// TwinCAT 3 PLC project MotionRail
// ProgramVersion: 3.1.4022.3
// libraries:
//   Tc2_MC2, * (Beckhoff Automation GmbH)
//   Tc2_Standard, * (Beckhoff Automation GmbH)
//   Tc2_System, * (Beckhoff Automation GmbH)
//   Tc3_Module, * (Beckhoff Automation GmbH)
// project tree:
//   / PlcTask.TcTTO
//   POUs/ FB_MicroStepCountTest.TcPOU, FB_MicroStepWalkTest.TcPOU, MAIN.TcPOU, FB_Tuning.TcPOU
// real-time tasks:
//   TASK PlcTask: cycle T#10ms, priority 20, ADS port 350
// motion (NC):
//   TASK NC-Task 1 SAF: cycle T#2ms, priority 4, ADS port 501
//   TASK NC-Task 1 SVB: cycle T#10ms, priority 8, ADS port 511
//   AXIS Axis 1 (id 1)
//     Dynamic: AccelerationMaximum=5, DecelerationMaximum=5, Acceleration=5, Deceleration=5, Jerk=5, DelayTime=0.008
//     Velo: Maximum=20
//     OtherSettings: AllowMotionCmdToSlave=true
//     encoder EncType=29
//       EncPara: ScaleFactorNumerator=5e-005, MaxCount=#xffffffff
//         SoftEndMinControl: Enable=true, Range=25
//         SoftEndMaxControl: Enable=true, Range=110
//         Inc: RefSoftSyncMask=#x0000ffff
//     drive DrvType=24
//       Analog: VeloReferenz=50, ScaleFactorActTorque=0.1
//       TimeComp: TaskDelayCycles=1
//     controller CtrType=2
//       CtrPara: PriorControlFactor=1
//         PosDiffControl: Range=0.1
//         PID: PosKp=20, PosExtKp=20, DeadBandPosition=0.000195
//         Observer: BandWidth=20
//   AXIS Axis 2 (id 2)
//     Dynamic: DelayTime=0.008
//     Velo: Maximum=5
//     OtherSettings: AllowMotionCmdToSlave=true
//     encoder EncType=4
//       EncPara: ScaleFactorNumerator=0.0001984375, MaxCount=#x0000ffff
//         Inc: RefMode=2, RefSoftSyncMask=#x0000ffff
//     drive DrvType=24
//       Analog: VeloReferenz=25.4, ScaleFactorActTorque=0.1
//       TimeComp: TaskDelayCycles=1
//     controller CtrType=1
//       CtrPara: PriorControlFactor=1
//         PosDiffControl: Range=0.635
//         Observer: BandWidth=20
//   AXIS Axis 3 (id 3)
//     Dynamic: DelayTime=0.008
//     Velo: Maximum=5
//     OtherSettings: AllowMotionCmdToSlave=true
//     encoder EncType=4
//       EncPara: ScaleFactorNumerator=0.0001984375, MaxCount=#x0000ffff
//         Inc: RefSoftSyncMask=#x0000ffff
//     drive DrvType=24
//       Analog: VeloReferenz=24.80437, ScaleFactorActTorque=0.1
//       TimeComp: TaskDelayCycles=1
//     controller CtrType=1
//       CtrPara: PriorControlFactor=1
//         PosDiffControl: Range=0.635
//         Observer: BandWidth=20
//   AXIS Axis 4 (id 4)
//     Dynamic: AccelerationMaximum=1000, DecelerationMaximum=1000, Acceleration=10, Deceleration=10, Jerk=100, DelayTime=0.008
//     Velo: RefSearch=1, RefSync=1, SlowManual=5, FastManual=5, Maximum=9
//     TargetPosControl: Range=0.001, Time=0.2
//     OtherSettings: AllowMotionCmdToSlave=true, PulseDistancePos=2, PulseDistanceNeg=2
//     encoder EncType=29
//       EncPara: ScaleFactorNumerator=5e-005, MaxCount=#xffffffff, ReferenceSystem=1
//         SoftEndMinControl: Enable=true, Range=5
//         SoftEndMaxControl: Enable=true, Range=60
//         Inc: RefSoftSyncMask=#x0000ffff
//     drive DrvType=24
//       Analog: VeloReferenz=25.4, ScaleFactorActTorque=0.1
//       TimeComp: TaskDelayCycles=1
//     controller CtrType=2
//       CtrPara: PriorControlFactor=1
//         PosDiffControl: Range=0.1
//         PID: PosKp=20, PosExtKp=5, DeadBandPosition=0.0001
//         Observer: BandWidth=20
// I/O:
//   DEVICE Device 1 (EtherCAT), AmsNetId 5.54.18.124.2.1
//     Term 1 (EK1200) [EK1200-5000 EtherCAT Power supply (2A E-Bus)]
//       Term 2 (EL7041) [EL7041 1Ch. Stepper motor output stage (50V, 5A)]
//       Term 3 (EL1004) [EL1004 4Ch. Dig. Input 24V, 3ms]
//       Term 4 (EL2008) [EL2008 8Ch. Dig. Output 24V, 0.5A]
//       Term 5 (EL5042) [EL5042 2Ch. BiSS-C Encoder]
//       Term 6 (EL7031) [EL7031 1Ch. Stepper motor output stage (24V, 1.5A)]
//       Term 7 (EL6001) [EL6001 Interface (RS232)]
//       Term 8 (EL7041-1000) [EL7041-1000 1Ch. Stepper motor output stage (50V, 5A, standard)]
//       Term 9 (EL5042) [EL5042 2Ch. BiSS-C Encoder]
//       Term 10 (EL7041) [EL7041 1Ch. Stepper motor output stage (50V, 5A)]
//       Term 11 (EL5042) [EL5042 2Ch. BiSS-C Encoder]
//       Term 12 (EL9011)
// variable links:
//   (this object) <-> Device 1 (EtherCAT)/Term 1 (EK1200)/Term 2 (EL7041)
//     Drive/Inputs/In/nState1 @bit 3 <-> STM Status/Status/Error
//     Drive/Inputs/In/nState1 @bit 5 <-> STM Status/Status/Moving negative
//     Drive/Inputs/In/nState1 @bit 4 <-> STM Status/Status/Moving positive
//     Drive/Inputs/In/nState1 @bit 1 <-> STM Status/Status/Ready
//     Drive/Inputs/In/nState1 <-> STM Status/Status/Ready to enable
//     Drive/Inputs/In/nState1 @bit 6 <-> STM Status/Status/Torque reduced
//     Drive/Inputs/In/nState1 @bit 2 <-> STM Status/Status/Warning
//     Drive/Inputs/In/nState2 @bit 3 <-> STM Status/Status/Digital input 1
//     Drive/Inputs/In/nState2 @bit 4 <-> STM Status/Status/Digital input 2
//     Drive/Inputs/In/nState4 @bit 1 <-> WcState/InputToggle
//     Drive/Inputs/In/nState4 <-> WcState/WcState
//     Drive/Outputs/Out/nCtrl1 <-> STM Control/Control/Enable
//     Drive/Outputs/Out/nCtrl1 @bit 2 <-> STM Control/Control/Reduce torque
//     Drive/Outputs/Out/nCtrl1 @bit 1 <-> STM Control/Control/Reset
//     Drive/Outputs/Out/nDataOut2[0] <-> STM Velocity/Velocity
//   (this object) <-> Device 1 (EtherCAT)/Term 1 (EK1200)/Term 5 (EL5042)
//     Enc/Inputs/In/nComState @bit 1 <-> WcState/InputToggle
//     Enc/Inputs/In/nComState <-> WcState/WcState
//     Enc/Inputs/In/nDataIn1 <-> FB Inputs Channel 1/Position
//     Enc/Inputs/In/nState1 @bit 12 <-> FB Inputs Channel 1/Status/Diag
//     Enc/Inputs/In/nState1 @bit 1 <-> FB Inputs Channel 1/Status/Error
//     Enc/Inputs/In/nState1 @bit 14 <-> FB Inputs Channel 1/Status/Input cycle counter
//     Enc/Inputs/In/nState1 @bit 2 <-> FB Inputs Channel 1/Status/Ready
//     Enc/Inputs/In/nState1 @bit 13 <-> FB Inputs Channel 1/Status/TxPDO State
//     Enc/Inputs/In/nState1 <-> FB Inputs Channel 1/Status/Warning
//   (this object) <-> Device 1 (EtherCAT)/Term 1 (EK1200)/Term 6 (EL7031)
//     Drive/Inputs/In/nState1 @bit 3 <-> STM Status/Status/Error
//     Drive/Inputs/In/nState1 @bit 5 <-> STM Status/Status/Moving negative
//     Drive/Inputs/In/nState1 @bit 4 <-> STM Status/Status/Moving positive
//     Drive/Inputs/In/nState1 @bit 1 <-> STM Status/Status/Ready
//     Drive/Inputs/In/nState1 <-> STM Status/Status/Ready to enable
//     Drive/Inputs/In/nState1 @bit 6 <-> STM Status/Status/Torque reduced
//     Drive/Inputs/In/nState1 @bit 2 <-> STM Status/Status/Warning
//     Drive/Inputs/In/nState2 @bit 3 <-> STM Status/Status/Digital input 1
//     Drive/Inputs/In/nState2 @bit 4 <-> STM Status/Status/Digital input 2
//     Drive/Inputs/In/nState2 @bit 5 <-> STM Status/Status/Sync error
//     Drive/Inputs/In/nState2 @bit 7 <-> STM Status/Status/TxPDO Toggle
//     Drive/Inputs/In/nState4 @bit 1 <-> WcState/InputToggle
//     Drive/Inputs/In/nState4 <-> WcState/WcState
//     Drive/Outputs/Out/nCtrl1 <-> STM Control/Control/Enable
//     Drive/Outputs/Out/nCtrl1 @bit 2 <-> STM Control/Control/Reduce torque
//     Drive/Outputs/Out/nCtrl1 @bit 1 <-> STM Control/Control/Reset
//     Drive/Outputs/Out/nDataOut2[0] <-> STM Velocity/Velocity
//     Enc/Inputs/In/nDataIn1[0] <-> ENC Status compact/Counter value
//     Enc/Inputs/In/nDataIn2[0] <-> ENC Status compact/Latch value
//     Enc/Inputs/In/nState1 @bit 4 <-> ENC Status compact/Status/Counter overflow
//     Enc/Inputs/In/nState1 @bit 3 <-> ENC Status compact/Status/Counter underflow
//     Enc/Inputs/In/nState1 @bit 1 <-> ENC Status compact/Status/Latch extern valid
//     Enc/Inputs/In/nState1 @bit 2 <-> ENC Status compact/Status/Set counter done
//     Enc/Inputs/In/nState2 @bit 4 <-> ENC Status compact/Status/Status of extern latch
//     Enc/Inputs/In/nState2 @bit 5 <-> ENC Status compact/Status/Sync error
//     Enc/Inputs/In/nState2 @bit 7 <-> ENC Status compact/Status/TxPDO Toggle
//     Enc/Inputs/In/nState4 @bit 1 <-> WcState/InputToggle
//     Enc/Inputs/In/nState4 <-> WcState/WcState
//     Enc/Outputs/Out/nCtrl1 @bit 3 <-> ENC Control compact/Control/Enable latch extern on negative edge
//     Enc/Outputs/Out/nCtrl1 @bit 1 <-> ENC Control compact/Control/Enable latch extern on positive edge
//     Enc/Outputs/Out/nCtrl1 @bit 2 <-> ENC Control compact/Control/Set counter
//     Enc/Outputs/Out/nDataOut1[0] <-> ENC Control compact/Set counter value
//   (this object) <-> Device 1 (EtherCAT)/Term 1 (EK1200)/Term 8 (EL7041-1000)
//     Drive/Inputs/In/nState1 @bit 3 <-> STM Status/Status/Error
//     Drive/Inputs/In/nState1 @bit 5 <-> STM Status/Status/Moving negative
//     Drive/Inputs/In/nState1 @bit 4 <-> STM Status/Status/Moving positive
//     Drive/Inputs/In/nState1 @bit 1 <-> STM Status/Status/Ready
//     Drive/Inputs/In/nState1 <-> STM Status/Status/Ready to enable
//     Drive/Inputs/In/nState1 @bit 6 <-> STM Status/Status/Torque reduced
//     Drive/Inputs/In/nState1 @bit 2 <-> STM Status/Status/Warning
//     Drive/Inputs/In/nState2 @bit 3 <-> STM Status/Status/Digital input 1
//     Drive/Inputs/In/nState2 @bit 4 <-> STM Status/Status/Digital input 2
//     Drive/Inputs/In/nState2 @bit 5 <-> STM Status/Status/Sync error
//     Drive/Inputs/In/nState2 @bit 7 <-> STM Status/Status/TxPDO Toggle
//     Drive/Inputs/In/nState4 @bit 1 <-> WcState/InputToggle
//     Drive/Inputs/In/nState4 <-> WcState/WcState
//     Drive/Outputs/Out/nCtrl1 <-> STM Control/Control/Enable
//     Drive/Outputs/Out/nCtrl1 @bit 2 <-> STM Control/Control/Reduce torque
//     Drive/Outputs/Out/nCtrl1 @bit 1 <-> STM Control/Control/Reset
//     Drive/Outputs/Out/nDataOut2[0] <-> STM Velocity/Velocity
//     Enc/Inputs/In/nDataIn1[0] <-> ENC Status compact/Counter value
//     Enc/Inputs/In/nDataIn2[0] <-> ENC Status compact/Latch value
//     Enc/Inputs/In/nState1 @bit 4 <-> ENC Status compact/Status/Counter overflow
//     Enc/Inputs/In/nState1 @bit 3 <-> ENC Status compact/Status/Counter underflow
//     Enc/Inputs/In/nState1 @bit 7 <-> ENC Status compact/Status/Extrapolation stall
//     Enc/Inputs/In/nState1 <-> ENC Status compact/Status/Latch C valid
//     Enc/Inputs/In/nState1 @bit 1 <-> ENC Status compact/Status/Latch extern valid
//     Enc/Inputs/In/nState1 @bit 2 <-> ENC Status compact/Status/Set counter done
//     Enc/Inputs/In/nState2 @bit 4 <-> ENC Status compact/Status/Status of extern latch
//     Enc/Inputs/In/nState2 <-> ENC Status compact/Status/Status of input A
//     Enc/Inputs/In/nState2 @bit 1 <-> ENC Status compact/Status/Status of input B
//     Enc/Inputs/In/nState2 @bit 2 <-> ENC Status compact/Status/Status of input C
//     Enc/Inputs/In/nState2 @bit 5 <-> ENC Status compact/Status/Sync error
//     Enc/Inputs/In/nState2 @bit 7 <-> ENC Status compact/Status/TxPDO Toggle
//     Enc/Inputs/In/nState4 @bit 1 <-> WcState/InputToggle
//     Enc/Inputs/In/nState4 <-> WcState/WcState
//     Enc/Outputs/Out/nCtrl1 <-> ENC Control compact/Control/Enable latch C
//     Enc/Outputs/Out/nCtrl1 @bit 3 <-> ENC Control compact/Control/Enable latch extern on negative edge
//     Enc/Outputs/Out/nCtrl1 @bit 1 <-> ENC Control compact/Control/Enable latch extern on positive edge
//     Enc/Outputs/Out/nCtrl1 @bit 2 <-> ENC Control compact/Control/Set counter
//     Enc/Outputs/Out/nDataOut1[0] <-> ENC Control compact/Set counter value
//   (this object) <-> Device 1 (EtherCAT)/Term 1 (EK1200)/Term 10 (EL7041)
//     Drive/Inputs/In/nState1 @bit 3 <-> STM Status/Status/Error
//     Drive/Inputs/In/nState1 @bit 5 <-> STM Status/Status/Moving negative
//     Drive/Inputs/In/nState1 @bit 4 <-> STM Status/Status/Moving positive
//     Drive/Inputs/In/nState1 @bit 1 <-> STM Status/Status/Ready
//     Drive/Inputs/In/nState1 <-> STM Status/Status/Ready to enable
//     Drive/Inputs/In/nState1 @bit 6 <-> STM Status/Status/Torque reduced
//     Drive/Inputs/In/nState1 @bit 2 <-> STM Status/Status/Warning
//     Drive/Inputs/In/nState2 @bit 3 <-> STM Status/Status/Digital input 1
//     Drive/Inputs/In/nState2 @bit 4 <-> STM Status/Status/Digital input 2
//     Drive/Inputs/In/nState2 @bit 5 <-> STM Status/Status/Sync error
//     Drive/Inputs/In/nState2 @bit 7 <-> STM Status/Status/TxPDO Toggle
//     Drive/Inputs/In/nState4 @bit 1 <-> WcState/InputToggle
//     Drive/Inputs/In/nState4 <-> WcState/WcState
//     Drive/Outputs/Out/nCtrl1 <-> STM Control/Control/Enable
//     Drive/Outputs/Out/nCtrl1 @bit 2 <-> STM Control/Control/Reduce torque
//     Drive/Outputs/Out/nCtrl1 @bit 1 <-> STM Control/Control/Reset
//     Drive/Outputs/Out/nDataOut2[0] <-> STM Velocity/Velocity
//   (this object) <-> Device 1 (EtherCAT)/Term 1 (EK1200)/Term 11 (EL5042)
//     Enc/Inputs/In/nComState @bit 1 <-> WcState/InputToggle
//     Enc/Inputs/In/nComState <-> WcState/WcState
//     Enc/Inputs/In/nDataIn1 <-> FB Inputs Channel 1/Position
//     Enc/Inputs/In/nState1 @bit 12 <-> FB Inputs Channel 1/Status/Diag
//     Enc/Inputs/In/nState1 @bit 1 <-> FB Inputs Channel 1/Status/Error
//     Enc/Inputs/In/nState1 @bit 14 <-> FB Inputs Channel 1/Status/Input cycle counter
//     Enc/Inputs/In/nState1 @bit 2 <-> FB Inputs Channel 1/Status/Ready
//     Enc/Inputs/In/nState1 @bit 13 <-> FB Inputs Channel 1/Status/TxPDO State
//     Enc/Inputs/In/nState1 <-> FB Inputs Channel 1/Status/Warning
//   MotionRail Instance <-> Device 1 (EtherCAT)/Term 1 (EK1200)/Term 10 (EL7041)
//     PlcTask Inputs/MAIN.bLimBwd4 <-> STM Status/Status/Digital input 2
//     PlcTask Inputs/MAIN.bLimFwd4 <-> STM Status/Status/Digital input 1
//   MotionRail Instance <-> Device 1 (EtherCAT)/Term 1 (EK1200)/Term 11 (EL5042)
//     PlcTask Inputs/MAIN.nRawCount4 <-> FB Inputs Channel 1/Position
//   MotionRail Instance <-> Device 1 (EtherCAT)/Term 1 (EK1200)/Term 2 (EL7041)
//     PlcTask Inputs/MAIN.bLimBwd1 <-> STM Status/Status/Digital input 2
//     PlcTask Inputs/MAIN.bLimFwd1 <-> STM Status/Status/Digital input 1
//   MotionRail Instance <-> Device 1 (EtherCAT)/Term 1 (EK1200)/Term 3 (EL1004)
//     PlcTask Inputs/MAIN.bHome1 <-> Channel 1/Input
//   MotionRail Instance <-> Device 1 (EtherCAT)/Term 1 (EK1200)/Term 4 (EL2008)
//     PlcTask Outputs/MAIN.bBrake1 <-> Channel 1/Output
//   MotionRail Instance <-> Device 1 (EtherCAT)/Term 1 (EK1200)/Term 5 (EL5042)
//     PlcTask Inputs/MAIN.fEnc2Raw <-> FB Inputs Channel 2/Position
//     PlcTask Inputs/MAIN.nRawCount1 <-> FB Inputs Channel 1/Position
//     PlcTask Inputs/MAIN.nRawCount2 <-> FB Inputs Channel 2/Position
//   MotionRail Instance <-> Device 1 (EtherCAT)/Term 1 (EK1200)/Term 6 (EL7031)
//     PlcTask Inputs/MAIN.bLimBwd2 <-> STM Status/Status/Digital input 2
//     PlcTask Inputs/MAIN.bLimFwd2 <-> STM Status/Status/Digital input 1
//   MotionRail Instance <-> Device 1 (EtherCAT)/Term 1 (EK1200)/Term 8 (EL7041-1000)
//     PlcTask Inputs/MAIN.bLimBwd3 <-> STM Status/Status/Digital input 2
//     PlcTask Inputs/MAIN.bLimFwd3 <-> STM Status/Status/Digital input 1
//   MotionRail Instance <-> Device 1 (EtherCAT)/Term 1 (EK1200)/Term 9 (EL5042)
//     PlcTask Inputs/MAIN.nRawCount3 <-> FB Inputs Channel 1/Position
//   MotionRail Instance <-> NC-Task 1 SAF/Axes/Axis 1
//     PlcTask Inputs/MAIN.Axis1.NcToPlc <-> Outputs/ToPlc
//     PlcTask Outputs/MAIN.Axis1.PlcToNc <-> Inputs/FromPlc
//   MotionRail Instance <-> NC-Task 1 SAF/Axes/Axis 2
//     PlcTask Inputs/MAIN.Axis2.NcToPlc <-> Outputs/ToPlc
//     PlcTask Outputs/MAIN.Axis2.PlcToNc <-> Inputs/FromPlc
//   MotionRail Instance <-> NC-Task 1 SAF/Axes/Axis 3
//     PlcTask Inputs/MAIN.Axis3.NcToPlc <-> Outputs/ToPlc
//     PlcTask Outputs/MAIN.Axis3.PlcToNc <-> Inputs/FromPlc
//   MotionRail Instance <-> NC-Task 1 SAF/Axes/Axis 4
//     PlcTask Inputs/MAIN.Axis4.NcToPlc <-> Outputs/ToPlc
//     PlcTask Outputs/MAIN.Axis4.PlcToNc <-> Inputs/FromPlc

CONFIGURATION MotionRail
    RESOURCE PLC ON TwinCAT3
        TASK PlcTask(INTERVAL := T#10ms, PRIORITY := 20);
        PROGRAM MAIN WITH PlcTask : MAIN;
    END_RESOURCE
END_CONFIGURATION

// ---- POUs/MAIN.TcPOU
PROGRAM MAIN
VAR
	Axis1: AXIS_REF;
	fbPower1: MC_POWER;
	bEnable1: BOOL := FALSE;
	bLimFwd1 AT %I*: BOOL;
	bLimBwd1 AT %I*: BOOL;
	bHome1 AT %I*: BOOL;
	bBrake1 AT %Q*: BOOL;
	fDeadband1: LREAL;
	fInvDeadband1: LREAL;
	nRawCount1 AT %I*: ULINT;
	
	Axis2: AXIS_REF;
	fbPower2: MC_POWER;
	bEnable2: BOOL := FALSE;
	bLimFwd2 AT %I*: BOOL;
	bLimBwd2 AT %I*: BOOL;
	bBrake2 AT %Q*: BOOL;
	fEnc2Raw AT %I*: LREAL;
	fDeadband2: LREAL;
	fInvDeadband2: LREAL;	
	nRawCount2 AT %I*: ULINT;
	
	Axis3: AXIS_REF;
	fbPower3: MC_POWER;
	bEnable3: BOOL := FALSE;
	bLimFwd3 AT %I*: BOOL;
	bLimBwd3 AT %I*: BOOL;
	bBrake3 AT %Q*: BOOL;
	fDeadband3: LREAL;
	fInvDeadband3: LREAL;
	nRawCount3 AT %I*: ULINT;
	
	Axis4: AXIS_REF;
	fbPower4: MC_POWER;
	bEnable4: BOOL := FALSE;
	bLimFwd4 AT %I*: BOOL;
	bLimBwd4 AT %I*: BOOL;
	bBrake4 AT %Q*: BOOL;
	fDeadband4: LREAL;
	fInvDeadband4: LREAL;
	nRawCount4 AT %I*: ULINT;
	
	bRefZero: BOOL;

	bDoTest: BOOL := FALSE;
	fbMicroWalkTest: FB_MicroStepWalkTest;
END_VAR

// Axis 1 is the standard circular motor connector + renishaw default pinout on the first channel of the first 5042
Axis1.ReadStatus();
fbPower1(Axis:=Axis1,
	Enable:=bEnable1,
	Enable_Positive:=bLimFwd1 OR TRUE,
	Enable_Negative:=bLimBwd1);
bBrake1 := Axis1.Status.ControlLoopClosed;
fDeadband1 := 0.000390625 / 2;
fInvDeadband1 := -fDeadband1;

// Axis 2 is the all-in-one motor/encoder connector on the second channel of the first 5042
Axis2.ReadStatus();
fbPower2(Axis:=Axis2,
	Enable:=bEnable2,
	Enable_Positive:=NOT bLimFwd2 OR TRUE,
	Enable_Negative:=NOT bLimBwd2 OR TRUE);
bBrake2 := Axis2.Status.ControlLoopClosed;

// Axis 3 is the stage with the magnetic encoder going to the first channel of the second 5042
Axis3.ReadStatus();
fbPower3(Axis:=Axis3,
	Enable:=bEnable3,
	Enable_Positive:=NOT bLimFwd3 OR TRUE,
	Enable_Negative:=NOT bLimBwd3 OR TRUE);
bBrake3 := Axis3.Status.ControlLoopClosed;

// Axis 4 is Alex's stage, going to the 4th drive and into the first channel of the third 5042
Axis4.ReadStatus();
fbPower4(Axis:=Axis4,
	Enable:=bEnable4,
	Enable_Positive:=NOT bLimFwd4 OR TRUE,
	Enable_Negative:=NOT bLimBwd4 OR TRUE);
bBrake4 := Axis4.Status.ControlLoopClosed;
fDeadband4 := 0.0001984375 / 2;
fInvDeadband4 := -1 * fDeadband4;

fbMicroWalkTest(bExecute:=bDoTest,
	nSteps:=1000,
	fDeadband:=fDeadband4 + 0.000025,
	fLowerBound:=10,
	fUpperBound:=55,
	fVelocity:=1,
	tSettleTime:=T#5S,
	Axis:=Axis4);

END_PROGRAM

// ---- POUs/FB_MicroStepWalkTest.TcPOU
FUNCTION_BLOCK FB_MicroStepWalkTest
VAR_INPUT
	bExecute: BOOL;
	nSteps: UINT;
	fDeadband: LREAL;
	fLowerBound: LREAL;
	fUpperBound: LREAL;
	fVelocity: LREAL;
	tSettleTime: TIME;
END_VAR
VAR_OUTPUT
	nGood: UINT;
	nBad: UINT;
	fPercent: LREAL;
	fAvgErr: LREAL;
	fMaxErr: LREAL;
	fMinErr: LREAL := 9001;
END_VAR
VAR_IN_OUT
	Axis: AXIS_REF;
END_VAR
VAR
	fbRand: DRAND;
	fbMove: MC_MoveAbsolute;
	fbSettleTimer: TON;
	bDoMove: BOOL;
	fGoal: LREAL;
	fStepErr: LREAL;
	fTotalErr: LREAL;
	nStepCounter: UINT;
END_VAR

// Moves to random positions and see how close we get to each one
// Pick random numbers from 0 to 1
fbRand(Seed:=UINT_TO_INT(nSteps));
// Latch a new random goal if we aren't moving
IF NOT bDoMove THEN
	fGoal := fbRand.Num * (fUpperBound - fLowerBound) + fLowerBound;
END_IF
// Motion FB
fbMove(Axis:=Axis,
	Execute:=bDoMove,
	Position:=fGoal,
	Velocity:=fVelocity);
// Settle time
fbSettleTimer(IN:=fbMove.Done,
	PT:=tSettleTime);
// Re-enable the move for next cycle
bDoMove := bExecute AND nStepCounter < nSteps;
// Check results
IF fbSettleTimer.Q THEN
	fStepErr := ABS(Axis.NcToPlc.PosDiff);
	IF fStepErr <= fDeadband THEN
		nGood := nGood + 1;
	ELSE
		nBad := nBad + 1;
	END_IF
	IF nGood + nBad > 0 THEN
		fPercent := 100 * nGood / (nGood + nBad);
	END_IF
	fTotalErr := fTotalErr + fStepErr;
	nStepCounter := nStepCounter + 1;
	IF nStepCounter > 0 THEN
		fAvgErr := fTotalErr / nStepCounter;
	END_IF
	IF fStepErr > fMaxErr THEN
		fMaxErr := fStepErr;
	END_IF
	IF fStepErr < fMinErr THEN
		fMinErr := fStepErr;
	END_IF
	// Reset the move block
	bDoMove := FALSE;
END_IF

END_FUNCTION_BLOCK

// ---- POUs/FB_MicroStepCountTest.TcPOU
FUNCTION_BLOCK FB_MicroStepCountTest
VAR_INPUT
	bExecute: BOOL;
	fStart: LREAL;
	fEnd: LREAL;
	fIncr: LREAL;
	fTheoryStep: LREAL;
END_VAR
VAR_OUTPUT
	bDone: BOOL;
	nPosCount: INT := -1;
	nTheoryCount: DINT;
	nSteps: INT := -1;
	nMissedSteps: INT;
	nMaxMissCombo: INT;
	fStepPercent: LREAL;
END_VAR
VAR_IN_OUT
	Axis: AXIS_REF;
END_VAR
VAR
	fbMoveStart: MC_MoveAbsolute;
	fbStep: MC_MoveRelative;
	fbSettleTimer: TON;
	bStarted: BOOL;
	bTimerLatch: BOOL;
	bDoStep: BOOL;
	nWaitCount: UINT;
	fLastPosition: LREAL;
	nMissCombo: INT;
	nOldTheoryCount: DINT;
END_VAR

// Goal: Move axis slightly, repeatedly, and see how many effective positions we have between two given positions.
// Works best if fIncr is greater than the encoder noise but less than the smallest theoretical step
fbMoveStart(Axis:=Axis,
	Execute:=bExecute AND NOT bStarted AND NOT bDone,
	Position:=fStart,
	Velocity:=1);
fbStep(Axis:=Axis,
	Execute:=bDoStep AND bStarted AND NOT bDone,
	Distance:=fIncr,
	Velocity:=1);
fbSettleTimer(IN:=fbMoveStart.Done OR fbStep.Done,
	PT:=T#2S);
IF fbSettleTimer.Q THEN
	IF NOT bStarted THEN
		bDoStep := TRUE;
	END_IF
	bStarted := TRUE;
	bTimerLatch := TRUE;
	nSteps := nSteps + 1;
	nOldTheoryCount := nTheoryCount;
	nTheoryCount := TRUNC((Axis.NcToPlc.ActPos - fStart)/fTheoryStep);
	IF Axis.NcToPlc.ActPos >= fLastPosition + fIncr THEN
		fLastPosition := Axis.NcToPlc.ActPos;
		nPosCount := nPosCount + 1;
		nMissCombo := 0;
	ELSIF nTheoryCount - nOldTheoryCount >= 1 THEN
		nMissedSteps := nMissedSteps + 1;
		nMissCombo := nMissCombo + 1;
		IF nMissCombo > nMaxMissCombo THEN
			nMaxMissCombo := nMissCombo;
		END_IF
	END_IF
	IF nTheoryCount > 0 THEN
		fStepPercent := 100 * nPosCount / nTheoryCount;
	END_IF
	IF fLastPosition >= fEnd THEN
		bDone := TRUE;
	END_IF
END_IF
IF bTimerLatch THEN
	bTimerLatch := bDoStep;
	bDoStep := NOT bDoStep;
END_IF

END_FUNCTION_BLOCK

// ---- POUs/FB_Tuning.TcPOU
FUNCTION_BLOCK FB_Tuning
VAR_INPUT
	bReset: BOOL;
	Axis: AXIS_REF;
	fDeadBand: LREAL;
	fEncRes: LREAL;
END_VAR
VAR_OUTPUT
	nSettleCount: UINT;
	nMaxSettleCount: UINT;
	fMaxFollowerError: LREAL;
	fMaxFollowerErrorCount: LREAL;
END_VAR
VAR
	
END_VAR

IF bReset THEN
	bReset := FALSE;
	nMaxSettleCount := 0;
	fMaxFollowerError := 0;
END_IF

Axis.ReadStatus();
// Settle time calculation
IF Axis.Status.NotMoving THEN
	IF ABS(Axis.NcToPlc.PosDiff) >= fDeadband THEN
		nSettleCount := nSettleCount + 1;
	END_IF
ELSE
	nSettleCount := 0;
END_IF
IF nSettleCount > nMaxSettleCount THEN
	nMaxSettleCount := nSettleCount;
END_IF

IF ABS(Axis.NcToPlc.PosDiff) > fMaxFollowerError THEN
	fMaxFollowerError := ABS(Axis.NcToPlc.PosDiff);
	fMaxFollowerErrorCount := fMaxFollowerError / fEncRes;
END_IF

END_FUNCTION_BLOCK
